FUNCTION isLeapYear : BOOL
VAR_INPUT
	Year : DINT;
END_VAR
VAR
END_VAR

isLeapYear := (year mod 4 = 0) and ((year mod 100 <> 0) or (year mod 400 = 0));

END_FUNCTION

(* stored: Version 1.1.0.1, ProductVersion 3.1.4024.12
   POU isLeapYear: Id {6342e5f8-04b6-4083-87c4-cf21a7f0562e}, SpecialFunc None *)
